Yaskawa INFORM job: R1_W31(0,0)_KM-OK.JBI

/JOB
//NAME R1_W31(0,0)_KM-OK
///FOLDERNAME KRIS-SCIANA
//POS
///NPOS 83,83,0,5,0,0
///TOOL 0
///POSTYPE PULSE
///PULSE
C00000=102126,18825,-41470,-65608,62226,36597
C00001=120339,23079,-19532,-81795,45939,24488
C00002=122189,67376,29099,-89357,43616,27152
C00003=121004,73460,34134,-89018,42790,27107
C00004=120543,75972,36286,-88933,42467,27118
C00005=120547,77449,38075,-89311,42453,27349
C00006=120543,75972,36286,-88933,42467,27118
C00007=123298,89224,41655,-76600,55308,25879
C00008=122969,89182,41601,-76463,55094,25842
C00009=119753,75938,36143,-88643,41920,27049
C00010=122777,93473,61536,-103228,51808,35130
C00011=122777,93480,60664,-102807,51709,34821
C00012=122056,93390,61432,-103190,51294,35173
C00013=122567,91090,59506,-103202,51654,35130
C00014=123870,85634,55138,-103330,52596,35092
C00015=125017,80252,31903,-67160,60858,30978
C00016=117036,62710,10886,-43727,44565,22201
C00017=116780,65499,14144,-43914,44034,22373
C00018=116807,67095,16018,-44174,43802,22532
C00019=116792,66139,14894,-44017,43942,22437
C00020=116001,66281,15059,-43374,43566,22196
C00021=115569,66368,15163,-43020,43361,22064
C00022=116269,62151,10243,-43005,44309,21910
C00023=122431,75509,15675,-42518,64116,27745
C00024=120732,80304,21747,-41899,62444,27757
C00025=114671,71267,10742,-25968,56507,20900
C00026=114705,72531,12271,-26076,56252,20980
C00027=120070,82309,24307,-41679,61753,27775
C00028=119168,83067,23974,-40915,61831,27344
C00029=118706,83060,23966,-40627,61642,27221
C00030=119100,72567,11015,-40039,63792,26480
C00031=117642,75656,20439,-40534,59943,27496
C00032=117664,77615,22834,-40721,59594,27660
C00033=117687,79508,25160,-40908,59252,27824
C00034=117671,78126,23459,-40772,59503,27706
C00035=119132,77976,23275,-41673,60150,28081
C00036=119142,79644,25327,-41833,59848,28225
C00037=118622,79686,25380,-41514,59616,28091
C00038=119921,74095,18542,-41829,61182,27971
C00039=123924,66248,9738,-82632,66113,-4047
C00040=107346,82155,44839,-154040,38328,-19284
C00041=107345,82085,44753,-154030,38313,-19290
C00042=107345,82076,44742,-154029,38311,-19290
C00043=105766,83514,47837,-160642,39177,-16573
C00044=107604,79582,41685,-153491,37881,-19627
C00045=107224,79409,41473,-153690,37712,-19470
C00046=105568,83740,56784,-163399,43972,-15262
C00047=105497,78624,56137,-164243,46040,-14757
C00048=105560,84741,63812,-164702,47541,-14457
C00049=107258,82886,61095,-119534,27741,-31091
C00050=106881,82684,60844,-119663,27474,-31013
C00051=105474,84388,47037,-160784,38039,-16850
C00052=106033,81368,44275,-160360,38056,-17159
C00053=105476,84004,47520,-161044,38496,-16704
C00054=107258,82806,60996,-119500,27732,-31108
C00055=106881,82604,60746,-119629,27464,-31030
C00056=105436,83815,56078,-163357,43478,-15326
C00057=105896,77477,52492,-163460,44578,-15292
C00058=105548,77217,41300,-160829,38199,-16836
C00059=105454,87496,42218,-158200,33862,-18277
C00060=107257,82726,60897,-119467,27722,-31125
C00061=106880,82524,60648,-119596,27455,-31047
C00062=105404,87275,42736,-158518,34238,-18103
C00063=105951,77674,28448,-155386,30954,-19846
C00064=105580,81535,40469,-159339,35706,-17678
C00065=105423,86018,45947,-160048,36632,-17264
C00066=107256,82646,60799,-119433,27713,-31142
C00067=106879,82445,60550,-119562,27446,-31064
C00068=109450,84136,37145,-137594,34929,-24129
C00069=110362,76235,26997,-134418,33961,-25844
C00070=110080,77212,36112,-139665,37329,-22921
C00071=109537,80538,40209,-140695,37705,-22256
C00072=107256,82566,60701,-119400,27704,-31159
C00073=106879,82365,60452,-119529,27437,-31081
C00074=109403,79512,43588,-142953,39606,-20934
C00075=109406,79203,47234,-144753,41465,-19866
C00076=111201,59852,25009,-141057,39445,-22245
C00077=109965,74870,36549,-141090,38405,-22076
C00078=109305,77783,39188,-141503,38190,-21764
C00079=109298,77272,44688,-144398,40977,-20067
C00080=111329,74932,41875,-142979,41525,-21122
C00081=48826,-12478,-44952,-111799,21990,-32460
C00082=48826,-14822,-37600,-124145,24456,-26472
BC00000=73931,604516,837779
BC00001=58622,631195,766983
BC00002=57127,633801,760067
BC00003=57127,633801,760067
BC00004=57127,633801,760067
BC00005=57127,633801,760067
BC00006=57127,633801,760067
BC00007=57127,633801,760067
BC00008=57127,633801,760067
BC00009=57127,633801,760067
BC00010=57127,633801,760067
BC00011=57127,633801,760067
BC00012=57127,633801,760067
BC00013=57127,633801,760067
BC00014=57127,633801,760067
BC00015=58679,633516,508320
BC00016=58679,633516,508320
BC00017=58679,633516,508320
BC00018=58679,633516,508320
BC00019=58679,633516,508320
BC00020=58679,633516,508320
BC00021=58679,633516,508320
BC00022=58679,633516,508320
BC00023=59666,633334,348167
BC00024=59666,633334,348167
BC00025=59666,633334,348167
BC00026=59666,633334,348167
BC00027=59666,633334,348167
BC00028=59666,633334,348167
BC00029=59666,633334,348167
BC00030=59666,633334,348167
BC00031=59666,633334,348167
BC00032=59666,633334,348167
BC00033=59666,633334,348167
BC00034=59666,633334,348167
BC00035=59666,633334,348167
BC00036=59666,633334,348167
BC00037=59666,633334,348167
BC00038=59666,633334,348167
BC00039=47019,643904,514312
BC00040=32533,656010,704605
BC00041=32553,626933,597054
BC00042=36828,621316,608367
BC00043=36826,621318,608359
BC00044=38538,619070,612892
BC00045=38538,619070,612892
BC00046=36828,621316,608366
BC00047=36828,621316,608367
BC00048=36827,621316,608366
BC00049=21216,642924,787864
BC00050=21216,642924,787864
BC00051=36828,621316,443157
BC00052=36828,621316,407024
BC00053=36828,621316,407024
BC00054=21238,643014,684592
BC00055=21238,643014,684592
BC00056=36828,621316,407024
BC00057=36828,621316,407024
BC00058=36828,621316,313069
BC00059=36828,621316,237457
BC00060=21261,643103,581320
BC00061=21261,643103,581320
BC00062=36828,621316,188211
BC00063=36828,621316,174572
BC00064=36828,621316,174572
BC00065=36828,621316,174572
BC00066=21284,643192,478048
BC00067=21284,643192,478048
BC00068=36828,620744,113964
BC00069=36828,620729,112363
BC00070=36827,620729,112362
BC00071=36828,620729,112363
BC00072=21306,643282,374776
BC00073=21306,643282,374776
BC00074=36828,620729,112363
BC00075=36828,620729,112363
BC00076=36828,620729,112363
BC00077=36828,620729,112363
BC00078=36828,620729,112363
BC00079=36828,620729,112363
BC00080=36828,620729,112880
BC00081=36828,620729,367967
BC00082=36828,620729,1041515
///POSTYPE BASE
///RECTAN
///RCONF 0,0,0,0,1,0,0,0,0,0,0,0,0,0,0,0,0,0,0,0,0,0,0,0
P00006=2.006,1.622,-0.565,0.0000,0.0000,0.0000
P00021=0.073,2.058,-0.109,0.0000,0.0000,0.0000
P00022=2.006,1.622,-0.565,0.0000,0.0000,0.0000
///RCONF 0,0,0,0,0,0,0,0,0,0,0,0,0,0,0,0,0,0,0,0,0,0,0,0
P00023=-2.957,-4.083,2.762,0.0000,0.0000,0.0000
P00024=-1.466,-0.226,-0.419,0.0000,0.0000,0.0000
//INST
///DATE 2025/02/26 13:47
///ATTR SC,RW
///GROUP1 RB1,BS1
NOP
SFTOF
MOVJ C00000 BC00000 VJ=100.00
MOVJ C00001 BC00001 VJ=100.00
MOVJ C00002 BC00002 VJ=100.00
MOVL C00003 BC00003 V=100.0
MOVL C00004 BC00004 V=60.0
REFP 3 C00005 BC00005
CALL JOB:SEARCH-R1
SET P021 P006
SFTON P021
MOVL C00006 BC00006 V=60.0
MOVL C00007 BC00007 V=60.0
REFP 3 C00008 BC00008
CALL JOB:SEARCH-R1
SET P021 P006
SFTON P021
MOVL C00009 BC00009 V=60.0
MOVL C00010 BC00010 V=60.0
REFP 3 C00011 BC00011
CALL JOB:SEARCH-R1
SET P021 P006
SFTON P021
MOVL C00012 BC00012 V=60.0
MOVL C00013 BC00013 V=100.0
MOVL C00014 BC00014 V=100.0
'Path S949 (for W950)
SFTOF
MOVJ C00015 BC00015 VJ=100.00
MOVL C00016 BC00016 V=100.0
MOVL C00017 BC00017 V=60.0
REFP 3 C00018 BC00018
CALL JOB:SEARCH-R1
SET P024 P006
SFTON P024
MOVL C00019 BC00019 V=100.0
MOVL C00020 BC00020 V=100.0
REFP 3 C00021 BC00021
CALL JOB:SEARCH-R1
SET P024 P006
SFTON P024
MOVL C00022 BC00022 V=100.0
SFTOF
MOVJ C00023 BC00023 VJ=100.00
COMM MOVL C00024 BC00024 V=100.0
COMM MOVL C00025 BC00025 V=60.0
COMM REFP 3 C00026 BC00026
COMM CALL JOB:SEARCH-R1
COMM SET P022 P006
COMM SFTON P022
COMM MOVL C00027 BC00027 V=60.0
COMM MOVL C00028 BC00028 V=60.0
COMM REFP 3 C00029 BC00029
COMM CALL JOB:SEARCH-R1
COMM SET P022 P006
COMM SFTON P022
COMM 'Path W950
COMM SFTOF
COMM MOVJ C00030 BC00030 VJ=100.00
COMM MOVL C00031 BC00031 V=400.0
COMM MOVL C00032 BC00032 V=100.0
COMM REFP 3 C00033 BC00033
COMM CALL JOB:SEARCH-R1
COMM SET P023 P006
COMM SFTON P023
COMM MOVL C00034 BC00034 V=100.0
COMM MOVL C00035 BC00035 V=400.0
COMM MOVL C00036 BC00036 V=100.0
COMM REFP 3 C00037 BC00037
COMM CALL JOB:SEARCH-R1
COMM SET P023 P006
COMM SFTON P023
COMM MOVL C00038 BC00038 V=400.0
SFTOF
MOVJ C00039 BC00039 VJ=100.00
MOVJ C00040 BC00040 VJ=100.00
SFTON P021
CALL JOB:COFNIJ_DRUT
MOVJ C00041 BC00041 VJ=100.00
MOVL C00042 BC00042 V=100.0
MOVL C00043 BC00043 V=100.0 PL=0
REFP 1 C00044 BC00044
REFP 2 C00045 BC00045
MACRO1 MJ#(0) ARGF10
ARCON
MOVL C00046 BC00046 V=10.8
ARCOF
MOVL C00047 BC00047 V=100.0
MOVL C00048 BC00048 V=100.0 PL=0
REFP 1 C00049 BC00049
REFP 2 C00050 BC00050
MACRO1 MJ#(0) ARGF10
ARCON
MOVL C00051 BC00051 V=10.8
ARCOF
MOVL C00052 BC00052 V=100.0
MOVL C00053 BC00053 V=100.0 PL=0
REFP 1 C00054 BC00054
REFP 2 C00055 BC00055
ARCON
MOVL C00056 BC00056 V=10.8
ARCOF
MOVL C00057 BC00057 V=100.0
MOVL C00058 BC00058 V=100.0
SFTON P024
MOVL C00059 BC00059 V=100.0 PL=0
REFP 1 C00060 BC00060
REFP 2 C00061 BC00061
ARCON
MOVL C00062 BC00062 V=10.8
ARCOF
MOVL C00063 BC00063 V=100.0
MOVL C00064 BC00064 V=100.0
MOVL C00065 BC00065 V=100.0 PL=0
REFP 1 C00066 BC00066
REFP 2 C00067 BC00067
ARCON
MOVL C00068 BC00068 V=10.8
ARCOF
MOVL C00069 BC00069 V=100.0
COMM MOVL C00070 BC00070 V=100.0
COMM SFTON P022
COMM MOVL C00071 BC00071 V=100.0 PL=0
COMM REFP 1 C00072 BC00072
COMM REFP 2 C00073 BC00073
COMM ARCON
COMM MOVL C00074 BC00074 V=10.8
COMM MOVL C00075 BC00075 V=10.8
COMM ARCOF
COMM MOVL C00076 BC00076 V=100.0
COMM JUMP *BP1
COMM MOVL C00077 BC00077 V=400.0
COMM SFTON P023
COMM MOVL C00078 BC00078 V=100.0 PL=0
COMM MACRO1 MJ#(0) ARGF9
COMM ARCON
COMM MOVL C00079 BC00079 V=10.8
COMM ARCOF
COMM MOVL C00080 BC00080 V=100.0
COMM *BP1
MOVL C00081 BC00081 V=1000.0
SFTOF
MOVJ C00082 BC00082 VJ=100.00
END
